FUNCTION POU : DINT
VAR_INPUT
	a: DINT;
	b: DINT;
END_VAR
VAR
END_VAR

Somma := a + b;

END_FUNCTION

(* stored: Version 1.1.0.1, ProductVersion 3.1.4024.12
   POU POU: Id {9f48191b-4191-4add-aa03-59f1ad082999}, SpecialFunc None *)
